FUNCTION F_GetGroupErrorData : ST_GroupErrorStruct
(**************************************************************************************
 * 	Application		:	BoxControl Framework
 *	Revision		:	$Revision: 404529 $
 *	Revision date	:	$Date: 2018-04-23 08:21:38 +0200 (Mo., 23 Apr 2018) $
 *	Last changed by	:	$Author: b7bolm $
 *	URL				:	$URL: http://almscdc.swisslog.com/repo/SWPD/Development/BoxControlFramework/20_Release/trunk/01_Software/BCF/BCF/JumpStart/20_Product/10_App/14_Groups/10_Lib/10_Conv/10_Functions/F_GetGroupErrorData.TcPOU $
 *
 *	Purpose			:	Return group error data
 *
 * ------------------------------------------------------------------------------------
 *	Copyright Swisslog [IP AG], Switzerland. All rights reserved.
 * 
 * ------------------------------------------------------------------------------------
 *	
 * 	Revision History: 
 *
 * 	VERSION			DATE			INITIALS			DESCRIPTION
 *	0.1				01.01.2001		swl					Example
 *
 **************************************************************************************)
VAR_INPUT
	eGroupNumber		: E_GroupNumber; // Group number
END_VAR


// Check if group number is valid
IF eGroupNumber > E_GroupNumber.G_BEGIN_GROUP AND
   eGroupNumber < E_GroupNumber.G_END_GROUP THEN

	// Check reference is valid
	IF __ISVALIDREF(GroupRegistry[eGroupNumber].rGroup) THEN
   		// Return error data
   		F_GetGroupErrorData := GroupRegistry[eGroupNumber].rGroup.GroupData.ErrorData;
	END_IF
END_IF

END_FUNCTION

(* stored: Version 1.1.0.1, ProductVersion 3.1.4022.12
   POU F_GetGroupErrorData: Id {ae81be2e-b348-4c30-9b11-8bb90eaed675}, SpecialFunc None *)
